FUNCTION TorrToMbarWithUnits : REAL
VAR_INPUT
    pressure_Torr : REAL;
END_VAR

TorrToMbarWithUnits := pressure_Torr * 1.3332236842;

END_FUNCTION

(* stored: Version 1.1.0.1, ProductVersion 3.1.4024.4
   POU TorrToMbarWithUnits: Id {a0e2930e-e3a4-487c-bff9-d1277265aa82}, SpecialFunc None *)
